(* PLC project machine, CODESYS STW CODESYS V3.5 SP11 - ESX-3CS, author isoloader *)
(* stored: creationDateTime 2026-05-19T11:34:01.4368509, version 0.1, modificationDateTime 2026-01-26T17:08:03, organization Isoloader *)
(* isoloader machine - common to both plc and secondary devices *)

(* {attribute 'qualified_only'} *)
TYPE t_pack_code : (cPackCodeNone := 0, cPackCodeSystem := 1, cPackCodeMovement := 2, cPackCodeReportable := 3, cPackCodeSpreader := 4, cPackCodeConfiguration := 5, cPackCodeUICommand := 6);
END_TYPE

FUNCTION_BLOCK PackChannelUInterface EXTENDS NonOperationalParticleSet
  VAR
    lPLCIncomingChannel : PackChannel;
    lPLCOutgoingChannel : PackChannel;
    lPLCOutgoingPacket : t_packet;
    lPLCIncomingPacket : t_packet;
    lDebugPack : BOOL := FALSE;
    lDebugUnpack : BOOL := FALSE;
    lDebugPackPacket : t_packet;
    lDebugUnpackPacket : t_packet;
    lPackTimer : t_timer;
    lPackSystem : REFERENCE TO PackSystem;
    lPackMovement : REFERENCE TO PackMovement;
    lPackReportable : REFERENCE TO PackReportable;
    lPackSpreader : REFERENCE TO PackSpreader;
    lPackUICommand : REFERENCE TO PackUICommand;
    lPackProvider : REFERENCE TO PackProvider;
  END_VAR

            ;
          

METHOD initialize
                  IF ((NOT(__ISVALIDREF(lPackSystem))) OR
	(NOT(__ISVALIDREF(lPackMovement))) OR
	(NOT(__ISVALIDREF(lPackReportable))) OR
	(NOT(__ISVALIDREF(lPackSpreader))) OR
	(NOT(__ISVALIDREF(lPackUICommand))) OR
	(NOT(__ISVALIDREF(lPackProvider)))) THEN
	gCodeErrorHandler(pMessage:=CONCAT('null reference in ',lIdentity));
END_IF
	
lPackTimer.lEnable := TRUE;
lPackTimer.lPeriod := T#60MS;
lPackTimer.initialize();

lPLCOutgoingChannel.register(ADR(lPackSystem)); // foobar particle reorganization
lPLCOutgoingChannel.register(ADR(lPackMovement));
lPLCOutgoingChannel.register(ADR(lPackReportable));
lPLCOutgoingChannel.register(ADR(lPackSpreader));
lPLCOutgoingChannel.initialize();

lPLCIncomingChannel.register(ADR(lPackUICommand));
lPLCIncomingChannel.initialize();

SUPER^.initialize();
                
END_METHOD

METHOD initializePackChannelUInterface
  VAR_INPUT
    packSystem : REFERENCE TO PackSystem;
    packMovement : REFERENCE TO PackMovement;
    packReportable : REFERENCE TO PackReportable;
    packSpreader : REFERENCE TO PackSpreader;
    packUICommand : REFERENCE TO PackUICommand;
    packProvider : REFERENCE TO PackProvider;
  END_VAR
                  lPackSystem REF= packSystem;
lPackMovement REF= packMovement;
lPackReportable REF= packReportable;
lPackSpreader REF= packSpreader;

lPackUICommand REF= packUICommand;

lPackProvider REF= packProvider;

                
END_METHOD

METHOD trigger : BOOL
  VAR_INPUT
    machineStateId : t_machine_state_id;
  END_VAR
                  lPLCOutgoingChannel.trigger(lPLCOutgoingPacket,machineStateId);

                
END_METHOD

PROPERTY PackMovement : REFERENCE TO PackMovement
GET
                    PackMovement ref= lPackMovement;
                  
END_GET
END_PROPERTY

PROPERTY PackReportable : REFERENCE TO PackReportable
GET
                    PackReportable ref= lPackReportable;
                  
END_GET
END_PROPERTY

PROPERTY PackSpreader : REFERENCE TO PackSpreader
GET
                    PackSpreader ref= lPackSpreader;
                  
END_GET
END_PROPERTY

PROPERTY PackSystem : REFERENCE TO PackSystem
GET
                    PackSystem ref= lPackSystem;
                  
END_GET
END_PROPERTY

PROPERTY PackUICommand : REFERENCE TO PackUICommand
GET
                    PackUICommand ref= lPackUICommand;
                  
END_GET
END_PROPERTY

PROPERTY TypeToken : t_medium_string
GET
                    TypeToken := 'PackChannelUI';
                  
END_GET
END_PROPERTY
END_FUNCTION_BLOCK

FUNCTION_BLOCK PackChannelUInterfacePLC EXTENDS PackChannelUInterface

            ;
          

METHOD pullPLCIncomingChannel : BOOL
                  pullPLCIncomingChannel := FALSE;

lPackProvider.pull();

IF (lPLCIncomingPacket.Byte1<>lPackProvider.PackIn1) THEN
	lPLCIncomingPacket.Byte1 := lPackProvider.PackIn1;
	lPLCIncomingPacket.Byte1 := lPLCIncomingPacket.Byte1 OR INT_TO_USINT(cPackCodeUICommand);
	gSystemPrimary.Active.registerUI();
	pullPLCIncomingChannel := TRUE;
END_IF

IF (lPLCIncomingPacket.Byte2<>lPackProvider.PackIn2) THEN
	lPLCIncomingPacket.Byte2 := lPackProvider.PackIn2;
	gSystemPrimary.Active.registerUI();
	pullPLCIncomingChannel := TRUE;
END_IF

IF (lPLCIncomingPacket.Byte3<>lPackProvider.PackIn3) THEN
	lPLCIncomingPacket.Byte3 := lPackProvider.PackIn3;
	gSystemPrimary.Active.registerUI();
	pullPLCIncomingChannel := TRUE;
END_IF

IF (lPLCIncomingPacket.Byte4<>lPackProvider.PackIn4) THEN
	lPLCIncomingPacket.Byte4 := lPackProvider.PackIn4;
	gSystemPrimary.Active.registerUI();
	pullPLCIncomingChannel := TRUE;
END_IF

IF (lPLCIncomingPacket.Byte5<>lPackProvider.PackIn5) THEN
	lPLCIncomingPacket.Byte5 := lPackProvider.PackIn5;
	gSystemPrimary.Active.registerUI();
	pullPLCIncomingChannel := TRUE;
END_IF

IF (lPLCIncomingPacket.Byte6<>lPackProvider.PackIn6) THEN
	lPLCIncomingPacket.Byte6 := lPackProvider.PackIn6;
	gSystemPrimary.Active.registerUI();
	pullPLCIncomingChannel := TRUE;
END_IF

IF (lPLCIncomingPacket.Byte7<>lPackProvider.PackIn7) THEN
	lPLCIncomingPacket.Byte7 := lPackProvider.PackIn7;
	gSystemPrimary.Active.registerUI();
	pullPLCIncomingChannel := TRUE;
END_IF

IF (lPLCIncomingPacket.Byte8<>lPackProvider.PackIn8) THEN
	lPLCIncomingPacket.Byte8 := lPackProvider.PackIn8;
	gSystemPrimary.Active.registerUI();
	pullPLCIncomingChannel := TRUE;
END_IF

                
END_METHOD

METHOD pushPLCOutgoingChannel
                  lPackProvider.PackOut1 := lPLCOutgoingPacket.Byte1;
lPackProvider.PackOut2 := lPLCOutgoingPacket.Byte2;
lPackProvider.PackOut3 := lPLCOutgoingPacket.Byte3;
lPackProvider.PackOut4 := lPLCOutgoingPacket.Byte4;
lPackProvider.PackOut5 := lPLCOutgoingPacket.Byte5;
lPackProvider.PackOut6 := lPLCOutgoingPacket.Byte6;
lPackProvider.PackOut7 := lPLCOutgoingPacket.Byte7;
lPackProvider.PackOut8 := lPLCOutgoingPacket.Byte8;

lPackProvider.push();

                
END_METHOD

METHOD operator
                  lPackTimer.operator();
IF ((NOT(lPackTimer.Enable)) OR (lPackTimer.Expired)) THEN
	lPackTimer.reset();

	lPLCOutgoingChannel.pack(lPLCOutgoingPacket);
	pushPLCOutgoingChannel();
			
	IF (lDebugPack) THEN
		lDebugPackPacket.copy(lPLCOutgoingPacket);
	END_IF
END_IF

IF (pullPLCIncomingChannel()) THEN
	IF (lDebugUnpack) THEN
		lDebugUnpackPacket.copy(lPLCIncomingPacket);
	END_IF

	lPLCIncomingChannel.unpack(lPLCIncomingPacket);
END_IF

                
END_METHOD
END_FUNCTION_BLOCK

FUNCTION_BLOCK PackMovement EXTENDS Packer
  VAR_INPUT
    lSteerStateA : t_adjust_state;
    lSteerStateB : t_adjust_state;
    lSteerStateC : t_adjust_state;
    lSteerStateD : t_adjust_state;
    lSteerTargetAngle : REAL;
    lSteerCurrentMode : t_steer_mode;
    lTravelActive : BOOL;
    lTravelVelocity : t_percentage;
    lLiftActive : BOOL;
    lLiftABPosition : t_percentage;
    lLiftCDPosition : t_percentage;
    lProgrammedMovementCurrent : t_prog_mov_code;
    lProgrammedMovementState : t_prog_mov_state;
  END_VAR

            
          

METHOD _unpack
  VAR_INPUT
    packet : REFERENCE TO t_packet;
  END_VAR
                  lSteerStateA := packet.unpackUSINT(5,3);
lSteerStateB := packet.unpackUSINT(8,3);
lSteerStateC := packet.unpackUSINT(11,3);
lSteerStateD := packet.unpackUSINT(14,3);

lSteerTargetAngle := AngleFromSINT(packet.unpackSINT(17,8));
lSteerCurrentMode := USINT_TO_INT(packet.unpackUSINT(25,4));

lTravelActive := packet.unpackBool(29);
lTravelVelocity :=  SignedPercentageFrom6bits(packet.unpackUSINT(30,6));

lLiftActive := packet.unpackBool(36);
lLiftABPosition := SignedPercentageFrom7bits(packet.unpackUSINT(37,7));
lLiftCDPosition := SignedPercentageFrom7bits(packet.unpackUSINT(44,7));

lProgrammedMovementCurrent := packet.unpackUSINT(51,5);
lProgrammedMovementState := packet.unpackUSINT(56,3);
                
END_METHOD

METHOD _pack
  VAR_INPUT
    packet : REFERENCE TO t_packet;
  END_VAR
                  packet.packUSINT(INT_TO_USINT(lSteerStateA),5,3);
packet.packUSINT(INT_TO_USINT(lSteerStateB),8,3);
packet.packUSINT(INT_TO_USINT(lSteerStateC),11,3);
packet.packUSINT(INT_TO_USINT(lSteerStateD),14,3);

packet.packSINT(AngleAsSINT(lSteerTargetAngle),17,8);
packet.packUSINT(INT_TO_USINT(lSteerCurrentMode),25,4);

packet.packBool(lTravelActive,29);
packet.packUSINT(SignedPercentageAs6bits(lTravelVelocity),30,6);

packet.packBool(lLiftActive,36);
packet.packUSINT(SignedPercentageAs7bits(lLiftABPosition),37,7);
packet.packUSINT(SignedPercentageAs7bits(lLiftCDPosition),44,7);

packet.packUSINT(INT_TO_USINT(lProgrammedMovementCurrent),51,5);
packet.packUSINT(INT_TO_USINT(lProgrammedMovementState),56,3);

                
END_METHOD

METHOD initialize
                  lCode := INT_TO_USINT(t_pack_code.cPackCodeMovement);

SUPER^.initialize();

                
END_METHOD
END_FUNCTION_BLOCK

FUNCTION_BLOCK PackReportable EXTENDS Packer
  VAR_INPUT
    lReportableA : t_ui_reportable;
    lReportableB : t_ui_reportable;
    lReportableC : t_ui_reportable;
    lReportableD : t_ui_reportable;
  END_VAR

            
          

METHOD _unpack
  VAR_INPUT
    packet : REFERENCE TO t_packet;
  END_VAR
  VAR
    b : BOOL;
  END_VAR
                  IF (packet.unpackBool(5)) THEN
	lReportableA.valid := TRUE;
	lReportableA.state := packet.unpackUSINT(6,8);
ELSE
	lReportableA.event := packet.unpackUSINT(6,8);
	IF (lReportableA.event=cECNone) THEN
		lReportableA.valid := FALSE;
		lReportableB.valid := FALSE;
		lReportableC.valid := FALSE;
		lReportableD.valid := FALSE;
		
		RETURN;				
	END_IF
	lReportableA.valid := TRUE;
END_IF
lReportableA.active := packet.unpackBool(14);
lReportableA.subsystem := packet.unpackUSINT(15,5);

IF (packet.unpackBool(20)) THEN
	lReportableB.valid := TRUE;
	lReportableB.state := packet.unpackUSINT(21,8);
ELSE
	lReportableB.event := packet.unpackUSINT(21,8);	
	IF (lReportableB.event=cECNone) THEN
		lReportableB.valid := FALSE;
		lReportableC.valid := FALSE;
		lReportableD.valid := FALSE;
		
		RETURN;				
	END_IF
	lReportableB.valid := TRUE;
END_IF
lReportableB.active := packet.unpackBool(29);
lReportableB.subsystem := packet.unpackUSINT(30,5);

IF (packet.unpackBool(35)) THEN
	lReportableC.valid := TRUE;
	lReportableC.state := packet.unpackUSINT(36,8);
ELSE
	lReportableC.event := packet.unpackUSINT(36,8);	
	IF (lReportableC.event=cECNone) THEN
		lReportableC.valid := FALSE;
		lReportableD.valid := FALSE;
		
		RETURN;				
	END_IF
	lReportableC.valid := TRUE;
END_IF
lReportableC.active := packet.unpackBool(44);
lReportableC.subsystem := packet.unpackUSINT(45,5);

IF (packet.unpackBool(50)) THEN
	lReportableD.valid := TRUE;
	lReportableD.state := packet.unpackUSINT(51,8);
ELSE
	lReportableD.event := packet.unpackUSINT(51,8);	
	IF (lReportableD.event=cECNone) THEN
		lReportableD.valid := FALSE;
		
		RETURN;				
	END_IF
	lReportableD.valid := TRUE;
END_IF
lReportableD.active := packet.unpackBool(59);
lReportableD.subsystem := packet.unpackUSINT(60,5);

                
END_METHOD

METHOD _pack
  VAR_INPUT
    packet : REFERENCE TO t_packet;
  END_VAR
                  IF (NOT(lReportableA.valid)) THEN
	RETURN;
END_IF
	
IF (lReportableA.event=cECNone) THEN
	packet.packBool(TRUE,5);
	packet.packUSINT(INT_TO_USINT(lReportableA.state),6,8);
ELSE
	packet.packBool(FALSE,5);
	packet.packUSINT(INT_TO_USINT(lReportableA.event),6,8);
END_IF
packet.packBool(lReportableA.active,14);
packet.packUSINT(INT_TO_USINT(lReportableA.subsystem),15,5);

IF (NOT(lReportableB.valid)) THEN
	RETURN;
END_IF

IF (lReportableB.event=cECNone) THEN
	packet.packBool(TRUE,20);
	packet.packUSINT(INT_TO_USINT(lReportableB.state),21,8);
ELSE
	packet.packBool(FALSE,20);
	packet.packUSINT(INT_TO_USINT(lReportableB.event),21,8);
END_IF
packet.packBool(lReportableB.active,29);
packet.packUSINT(INT_TO_USINT(lReportableB.subsystem),30,5);

IF (NOT(lReportableC.valid)) THEN
	RETURN;
END_IF

IF (lReportableC.event=cECNone) THEN
	packet.packBool(TRUE,35);
	packet.packUSINT(INT_TO_USINT(lReportableC.state),36,8);
ELSE
	packet.packBool(FALSE,35);
	packet.packUSINT(INT_TO_USINT(lReportableC.event),36,8);
END_IF
packet.packBool(lReportableC.active,44);
packet.packUSINT(INT_TO_USINT(lReportableC.subsystem),45,5);

IF (NOT(lReportableD.valid)) THEN
	RETURN;
END_IF

IF (lReportableD.event=cECNone) THEN
	packet.packBool(TRUE,50);
	packet.packUSINT(INT_TO_USINT(lReportableD.state),51,8);
ELSE
	packet.packBool(FALSE,50);
	packet.packUSINT(INT_TO_USINT(lReportableD.event),51,8);
END_IF
packet.packBool(lReportableD.active,59);
packet.packUSINT(INT_TO_USINT(lReportableD.subsystem),60,5);

                
END_METHOD

METHOD initialize
                  lCode := INT_TO_USINT(t_pack_code.cPackCodeReportable);

SUPER^.initialize();

                
END_METHOD

METHOD reset
                  SUPER^.reset();

lReportableA.valid := FALSE;
lReportableB.valid := FALSE;
lReportableC.valid := FALSE;
lReportableD.valid := FALSE;
                
END_METHOD
END_FUNCTION_BLOCK

FUNCTION_BLOCK PackSpreader EXTENDS Packer
  VAR_INPUT
    lSideShiftActive : BOOL;
    lTwistlocksState : t_lock_state;
    lStateA : t_lock_state;
    lLoweredA : BOOL;
    lStateB : t_lock_state;
    lLoweredB : BOOL;
    lStateC : t_lock_state;
    lLoweredC : BOOL;
    lStateD : t_lock_state;
    lLoweredD : BOOL;
    lExtensionState : t_spreader_extension_state;
    lSpreaderOperationEnabled : BOOL;
    lSpreaderOperationActive : BOOL;
    lSpreaderConfigurationOptionEnabled : BOOL;
    lSpreaderConfigurationEnabled : BOOL;
    lSpreaderConfigurationActive : BOOL;
    lSpreaderConfigurationExtending : BOOL;
    lSpreaderConfigurationRetracting : BOOL;
    lTopbeamActive : BOOL;
    lTopbeamABPosition : t_percentage;
    lTopbeamCDPosition : t_percentage;
  END_VAR

            
          

METHOD _unpack
  VAR_INPUT
    packet : REFERENCE TO t_packet;
  END_VAR
                  lSideShiftActive := packet.unpackBool(5);

lTwistlocksState := packet.unpackUSINT(6,2);

lStateA := packet.unpackUSINT(8,2);
lLoweredA := packet.unpackBool(10);
lStateB := packet.unpackUSINT(11,2);
lLoweredB := packet.unpackBool(13);
lStateC := packet.unpackUSINT(14,2);
lLoweredC := packet.unpackBool(16);
lStateD := packet.unpackUSINT(17,2);
lLoweredD := packet.unpackBool(19);

lExtensionState := packet.unpackUSINT(20,2);
lSpreaderOperationEnabled := packet.unpackBool(22);
lSpreaderOperationActive := packet.unpackBool(23);

lSpreaderConfigurationOptionEnabled := packet.unpackBool(24);
lSpreaderConfigurationEnabled := packet.unpackBool(25);
lSpreaderConfigurationActive := packet.unpackBool(26);
lSpreaderConfigurationExtending := packet.unpackBool(27);
lSpreaderConfigurationRetracting := packet.unpackBool(28);

lTopbeamActive := packet.unpackBool(29);
lTopbeamABPosition := SignedPercentageFrom7bits(packet.unpackUSINT(30,7));
lTopbeamCDPosition := SignedPercentageFrom7bits(packet.unpackUSINT(37,7));


                
END_METHOD

METHOD _pack
  VAR_INPUT
    packet : REFERENCE TO t_packet;
  END_VAR
                  packet.packBool(lSideShiftActive,5);

//6-32 27 bits

packet.packUSINT(INT_TO_USINT(lTwistlocksState),6,2);

packet.packUSINT(INT_TO_USINT(lStateA),8,2);
packet.packBool(lLoweredA,10);
packet.packUSINT(INT_TO_USINT(lStateB),11,2);
packet.packBool(lLoweredB,13);
packet.packUSINT(INT_TO_USINT(lStateC),14,2);
packet.packBool(lLoweredC,16);
packet.packUSINT(INT_TO_USINT(lStateD),17,2);
packet.packBool(lLoweredD,19);

packet.packUSINT(INT_TO_USINT(lExtensionState),20,2);
packet.packBool(lSpreaderOperationEnabled,22);
packet.packBool(lSpreaderOperationActive,23);

packet.packBool(lSpreaderConfigurationOptionEnabled,24);
packet.packBool(lSpreaderConfigurationEnabled,25);
packet.packBool(lSpreaderConfigurationActive,26);
packet.packBool(lSpreaderConfigurationExtending,27);
packet.packBool(lSpreaderConfigurationRetracting,28);

packet.packBool(lTopbeamActive,29);
packet.packUSINT(SignedPercentageAs7bits(lTopbeamABPosition),30,7);
packet.packUSINT(SignedPercentageAs7bits(lTopbeamCDPosition),37,7);


                
END_METHOD

METHOD initialize
                  lCode := INT_TO_USINT(t_pack_code.cPackCodeSpreader);

SUPER^.initialize();
                
END_METHOD
END_FUNCTION_BLOCK

FUNCTION_BLOCK PackSystem EXTENDS Packer
  VAR_INPUT
    lFunctionalMode : t_functional_mode;
    lToggle : BOOL;
    lSystemState : t_system_state;
    lOperatingMode : t_operating_mode;
    lSpeedModeSlow : BOOL;
    lLightStatus : BOOL;
    lUIReady : BOOL;
    lUIModeRequest : BOOL;
    lUIMode : t_ui_mode;
    lHours : UINT;
    lSOC : t_percentage;
    lCurrent : t_percentage;
    lInputMode : t_input_mode;
    lUIOrientation : t_ui_orientation;
    lAvailability : t_percentage;
  END_VAR
  VAR
    lOverrideSystemState : BOOL := FALSE;
    lOverrideSystemStateValue : t_system_state := cSystemStateOperational;
  END_VAR

            
          

METHOD _unpack
  VAR_INPUT
    packet : REFERENCE TO t_packet;
  END_VAR
                  lFunctionalMode := packet.unpackUSINT(5,3);
lToggle := packet.unpackBool(8);
lSystemState := packet.unpackUSINT(9,4);
lOperatingMode := packet.unpackUSINT(13,4);
lSpeedModeSlow := packet.unpackBool(17);
lLightStatus := packet.unpackBool(18);
lUIReady := packet.unpackBool(19);
lUIModeRequest := packet.unpackBool(20);
lUIMode := packet.unpackUSINT(21,2);
lHours := packet.unpackUINT(23,16);
lSOC := PercentageFrom7bits(packet.unpackUSINT(39,7));
lCurrent := SignedPercentageFrom8bits(packet.unpackUSINT(46,8));
lInputMode := packet.unpackUSINT(54,2);
lUIOrientation := packet.unpackUSINT(56,3);
lAvailability := PercentageFrom4bits(packet.unpackUSINT(59,4));

IF (lOverrideSystemState) THEN
	lSystemState := lOverrideSystemStateValue;
END_IF


                
END_METHOD

METHOD _pack
  VAR_INPUT
    packet : REFERENCE TO t_packet;
  END_VAR
                  packet.packUSINT(INT_TO_USINT(lFunctionalMode),5,3);
packet.packBool(lToggle,8);
packet.packUSINT(INT_TO_USINT(lSystemState),9,4);
packet.packUSINT(INT_TO_USINT(lOperatingMode),13,4);
packet.packBool(lSpeedModeSlow,17);
packet.packBool(lLightStatus,18);
packet.packBool(lUIReady,19);
packet.packBool(lUIModeRequest,20);
packet.packUSINT(INT_TO_USINT(lUIMode),21,2);
packet.packUINT(lHours,23,16);
packet.packUSINT(PercentageAs7bits(lSOC),39,7);
packet.packUSINT(SignedPercentageAs8bits(lCurrent),46,8);
packet.packUSINT(INT_TO_USINT(lInputMode),54,2);
packet.packUSINT(INT_TO_USINT(lUIOrientation),56,3);
packet.packUSINT(PercentageAs4bits(lAvailability),59,4);

                
END_METHOD

METHOD initialize
                  lCode := INT_TO_USINT(t_pack_code.cPackCodeSystem);

SUPER^.initialize();



                
END_METHOD
END_FUNCTION_BLOCK

FUNCTION_BLOCK PackUICommand EXTENDS Packer
  VAR_INPUT
    lUIModeResponse : BOOL;
    lUIEventCodeRequest : t_ui_event_code;
    lSteerModeRequest : t_steer_mode;
    lOperatingMethodRequest : t_operating_method;
    lFunctionalModeRequest : t_functional_mode;
    lInputModeRequest : t_input_mode;
    lUIOrientationRequest : t_ui_orientation;
    lAutomationRequest : t_prog_mov_code;
    lIsBeginner : BOOL;
    lOverride : BOOL;
    lReportableA : t_ui_reportable;
    lReportableB : t_ui_reportable;
  END_VAR
  VAR
    lTimer : t_timer;
  END_VAR

            
          

METHOD reset
                  SUPER^.reset();

lUIModeResponse := FALSE;
lUIEventCodeRequest := cUIEventCodeNone;
lSteerModeRequest := cSteerModeNone;
lOperatingMethodRequest := cOperatingMethodNone;
lFunctionalModeRequest := cFunctionalModeAny;
lInputModeRequest := cInputModeNone;
lAutomationRequest := cProgMovCodeNone;
lIsBeginner := FALSE;

lReportableA.valid := FALSE;
lReportableB.valid := FALSE;


                
END_METHOD

METHOD trigger : BOOL
  VAR_INPUT
    packet : REFERENCE TO t_packet;
    machineStateId : t_machine_state_id;
  END_VAR
                  trigger := TRUE;
(*
CASE machineStateId OF
	t_machine_state_id.cMSIdNone:
		RETURN;

	t_machine_state_id.cMSIdSteerModeRequest:
		lTimer.reset();		
		packet.packUSINT(INT_TO_USINT(lPackRadioDashboard.lSteerModeRequest),14,3);
		RETURN;

	t_machine_state_id.cMSIdSteerModeRequest4WS:
		lTimer.reset();		
		packet.packUSINT(INT_TO_USINT(t_steer_mode.cSteerMode4WS),14,3);
		RETURN;

	t_machine_state_id.cMSIdSteerModeRequestLateral:
		lTimer.reset();		
		packet.packUSINT(INT_TO_USINT(t_steer_mode.cSteerModeLateral),14,3);
		RETURN;

	t_machine_state_id.cMSIdSteerModeRequestCarousel:
		lTimer.reset();		
		packet.packUSINT(INT_TO_USINT(t_steer_mode.cSteerModeCarousel),14,3);
		RETURN;

	
	t_machine_state_id.cMSIdToggleLightsRequest:
		lTimer.reset();
		packet.packUSINT(INT_TO_USINT(t_ui_event_code.cUIEventCodeToggleLights),8,6);
		RETURN;
	
	t_machine_state_id.cMSIdRadioModeResponse:
		lTimer.reset();
		packet.packUSINT(INT_TO_USINT(t_ui_event_code.cUIEventCodeUIModeResponse),8,6);		
		RETURN;
		
	t_machine_state_id.cMSIdOperatingModeRequest:
		lTimer.reset();		
		packet.packUSINT(INT_TO_USINT(lPackRadioDashboard.lOperatingMethodRequest),17,3);	
		RETURN;

	t_machine_state_id.cMSIdSpreaderTelescopingExtensionStateRequest6m:
		lTimer.reset();		
		packet.packUSINT(INT_TO_USINT(t_spreader_extension_state.cSpreaderExtensionState6m),20,2);
		RETURN;
	
	t_machine_state_id.cMSIdSpreaderTelescopingExtensionStateRequest9m:
		lTimer.reset();		
		packet.packUSINT(INT_TO_USINT(t_spreader_extension_state.cSpreaderExtensionState9m),20,2);
		RETURN;
		
	t_machine_state_id.cMSIdSpreaderTelescopingExtensionStateRequest12m:
		lTimer.reset();		
		packet.packUSINT(INT_TO_USINT(t_spreader_extension_state.cSpreaderExtensionState12m),20,2);
		RETURN;

	t_machine_state_id.cMSIdSpreaderGrabArmsExtendABRequest:
		lTimer.reset();		
		packet.packUSINT(INT_TO_USINT(t_spreader_extension_method.cSpreaderExtensionMethodABExtend),22,3);
		RETURN;

	t_machine_state_id.cMSIdSpreaderGrabArmsRetractABRequest:
		lTimer.reset();		
		packet.packUSINT(INT_TO_USINT(t_spreader_extension_method.cSpreaderExtensionMethodABRetract),22,3);	
		RETURN;

	t_machine_state_id.cMSIdSpreaderGrabArmsExtendCDRequest:
		lTimer.reset();		
		packet.packUSINT(INT_TO_USINT(t_spreader_extension_method.cSpreaderExtensionMethodCDExtend),22,3);	
		RETURN;

	t_machine_state_id.cMSIdSpreaderGrabArmsRetractCDRequest:
		lTimer.reset();		
		packet.packUSINT(INT_TO_USINT(t_spreader_extension_method.cSpreaderExtensionMethodCDRetract),22,3);		
		RETURN;
		
	t_machine_state_id.cMSIdLiftTopRequest:
		lTimer.reset();
		packet.packUSINT(INT_TO_USINT(t_ui_event_code.cUIEventCodeLiftTop),8,6);
		RETURN;	
		
END_CASE
*)
trigger := FALSE;

                
END_METHOD

METHOD _unpack
  VAR_INPUT
    packet : REFERENCE TO t_packet;
  END_VAR
                  lUIModeResponse := packet.unpackBool(5);
lUIEventCodeRequest := packet.unpackUSINT(6,6);
lSteerModeRequest := packet.unpackUSINT(12,3);
lOperatingMethodRequest := packet.unpackUSINT(15,3);
lFunctionalModeRequest := packet.unpackUSINT(18,3);
lInputModeRequest := packet.unpackUSINT(21,2);
lUIOrientationRequest := packet.unpackUSINT(23,3);
lAutomationRequest := packet.unpackUSINT(26,5);
lIsBeginner := packet.unpackBool(31);
lOverride := packet.unpackBool(32);

IF (packet.unpackBool(33)) THEN
	lReportableA.valid := TRUE;
	lReportableA.state := packet.unpackUSINT(34,8);
ELSE
	lReportableA.event := packet.unpackUSINT(34,8);
	IF (lReportableA.event=cECNone) THEN
		lReportableA.valid := FALSE;
		lReportableB.valid := FALSE;
		
		RETURN;				
	END_IF
	lReportableA.valid := TRUE;
END_IF
lReportableA.active := packet.unpackBool(42);
lReportableA.subsystem := packet.unpackUSINT(43,5);

IF (packet.unpackBool(49)) THEN
	lReportableB.valid := TRUE;
	lReportableB.state := packet.unpackUSINT(50,8);
ELSE
	lReportableB.event := packet.unpackUSINT(50,8);	
	IF (lReportableB.event=cECNone) THEN
		lReportableB.valid := FALSE;
		
		RETURN;				
	END_IF
	lReportableB.valid := TRUE;
END_IF
lReportableB.active := packet.unpackBool(58);
lReportableB.subsystem := packet.unpackUSINT(59,5);

                
END_METHOD

METHOD initialize
                  lCode := INT_TO_USINT(t_pack_code.cPackCodeUICommand);

SUPER^.initialize();

lTimer.initialize();
lTimer.Enable := TRUE;
lTimer.Period := T#60MS;


                
END_METHOD

METHOD _pack
  VAR_INPUT
    packet : REFERENCE TO t_packet;
  END_VAR
                  packet.packBool(lUIModeResponse,5);
packet.packUSINT(INT_TO_USINT(lUIEventCodeRequest),6,6);
packet.packUSINT(INT_TO_USINT(lSteerModeRequest),12,3);
packet.packUSINT(INT_TO_USINT(lOperatingMethodRequest),15,3);
packet.packUSINT(INT_TO_USINT(lFunctionalModeRequest),18,3);
packet.packUSINT(INT_TO_USINT(lInputModeRequest),21,2);
packet.packUSINT(INT_TO_USINT(lUIOrientationRequest),23,3);
packet.packUSINT(INT_TO_USINT(lAutomationRequest),26,5);
packet.packBool(lIsBeginner,31);
packet.packBool(lOverride,32);

IF (NOT(lReportableA.valid)) THEN
	RETURN;
END_IF
	
IF (lReportableA.event=cECNone) THEN
	packet.packBool(TRUE,33);
	packet.packUSINT(INT_TO_USINT(lReportableA.state),34,8);
ELSE
	packet.packBool(FALSE,33);
	packet.packUSINT(INT_TO_USINT(lReportableA.event),34,8);
END_IF
packet.packBool(lReportableA.active,42);
packet.packUSINT(INT_TO_USINT(lReportableA.subsystem),43,5);

IF (NOT(lReportableB.valid)) THEN
	RETURN;
END_IF
	
IF (lReportableB.event=cECNone) THEN
	packet.packBool(TRUE,49);
	packet.packUSINT(INT_TO_USINT(lReportableB.state),50,8);
ELSE
	packet.packBool(FALSE,49);
	packet.packUSINT(INT_TO_USINT(lReportableB.event),50,8);
END_IF
packet.packBool(lReportableB.active,58);
packet.packUSINT(INT_TO_USINT(lReportableB.subsystem),59,5);

                
END_METHOD
END_FUNCTION_BLOCK

FUNCTION_BLOCK PackProvider EXTENDS NonOperationalParticleSet
  VAR
    lPackIn1 : ValueObjectUSINTInputReferenceUSINT;
    lPackIn2 : ValueObjectUSINTInputReferenceUSINT;
    lPackIn3 : ValueObjectUSINTInputReferenceUSINT;
    lPackIn4 : ValueObjectUSINTInputReferenceUSINT;
    lPackIn5 : ValueObjectUSINTInputReferenceUSINT;
    lPackIn6 : ValueObjectUSINTInputReferenceUSINT;
    lPackIn7 : ValueObjectUSINTInputReferenceUSINT;
    lPackIn8 : ValueObjectUSINTInputReferenceUSINT;
    lPackOut1 : ValueObjectUSINTOutputReferenceUSINT;
    lPackOut2 : ValueObjectUSINTOutputReferenceUSINT;
    lPackOut3 : ValueObjectUSINTOutputReferenceUSINT;
    lPackOut4 : ValueObjectUSINTOutputReferenceUSINT;
    lPackOut5 : ValueObjectUSINTOutputReferenceUSINT;
    lPackOut6 : ValueObjectUSINTOutputReferenceUSINT;
    lPackOut7 : ValueObjectUSINTOutputReferenceUSINT;
    lPackOut8 : ValueObjectUSINTOutputReferenceUSINT;
  END_VAR

            ;
          

METHOD push
                  lPackOut1.operator();
lPackOut2.operator();
lPackOut3.operator();
lPackOut4.operator();
lPackOut5.operator();
lPackOut6.operator();
lPackOut7.operator();
lPackOut8.operator();

                
END_METHOD

METHOD pull
                  lPackIn1.operator();
lPackIn2.operator();
lPackIn3.operator();
lPackIn4.operator();
lPackIn5.operator();
lPackIn6.operator();
lPackIn7.operator();
lPackIn8.operator();

                
END_METHOD

METHOD initialize
                  lPackIn1.initializeValueObjectOp(NopSelf,'PackIn1','Packet 1 to master','',cValueStyleConfigurable);
lPackIn2.initializeValueObjectOp(NopSelf,'PackIn2','Packet 2 to master','',cValueStyleConfigurable);
lPackIn3.initializeValueObjectOp(NopSelf,'PackIn3','Packet 3 to master','',cValueStyleConfigurable);
lPackIn4.initializeValueObjectOp(NopSelf,'PackIn4','Packet 4 to master','',cValueStyleConfigurable);
lPackIn5.initializeValueObjectOp(NopSelf,'PackIn5','Packet 5 to master','',cValueStyleConfigurable);
lPackIn6.initializeValueObjectOp(NopSelf,'PackIn6','Packet 6 to master','',cValueStyleConfigurable);
lPackIn7.initializeValueObjectOp(NopSelf,'PackIn7','Packet 7 to master','',cValueStyleConfigurable);
lPackIn8.initializeValueObjectOp(NopSelf,'PackIn8','Packet 8 to master','',cValueStyleConfigurable);

lPackOut1.initializeValueObjectOp(NopSelf,'PackOut1','Packet 1 from master','',cValueStyleConfigurable);
lPackOut2.initializeValueObjectOp(NopSelf,'PackOut2','Packet 2 from master','',cValueStyleConfigurable);
lPackOut3.initializeValueObjectOp(NopSelf,'PackOut3','Packet 3 from master','',cValueStyleConfigurable);
lPackOut4.initializeValueObjectOp(NopSelf,'PackOut4','Packet 4 from master','',cValueStyleConfigurable);
lPackOut5.initializeValueObjectOp(NopSelf,'PackOut5','Packet 5 from master','',cValueStyleConfigurable);
lPackOut6.initializeValueObjectOp(NopSelf,'PackOut6','Packet 6 from master','',cValueStyleConfigurable);
lPackOut7.initializeValueObjectOp(NopSelf,'PackOut7','Packet 7 from master','',cValueStyleConfigurable);
lPackOut8.initializeValueObjectOp(NopSelf,'PackOut8','Packet 8 from master','',cValueStyleConfigurable);

SUPER^.initialize();
SubSystem := cSubsystemUInterface;

                
END_METHOD

METHOD initializePackProvider
  VAR_INPUT
    packIn1 : REFERENCE TO USINT;
    packIn2 : REFERENCE TO USINT;
    packIn3 : REFERENCE TO USINT;
    packIn4 : REFERENCE TO USINT;
    packIn5 : REFERENCE TO USINT;
    packIn6 : REFERENCE TO USINT;
    packIn7 : REFERENCE TO USINT;
    packIn8 : REFERENCE TO USINT;
    packOut1 : REFERENCE TO USINT;
    packOut2 : REFERENCE TO USINT;
    packOut3 : REFERENCE TO USINT;
    packOut4 : REFERENCE TO USINT;
    packOut5 : REFERENCE TO USINT;
    packOut6 : REFERENCE TO USINT;
    packOut7 : REFERENCE TO USINT;
    packOut8 : REFERENCE TO USINT;
  END_VAR
                  lPackIn1.InputReference REF= packIn1;
lPackIn2.InputReference REF= packIn2;
lPackIn3.InputReference REF= packIn3;
lPackIn4.InputReference REF= packIn4;
lPackIn5.InputReference REF= packIn5;
lPackIn6.InputReference REF= packIn6;
lPackIn7.InputReference REF= packIn7;
lPackIn8.InputReference REF= packIn8;

lPackOut1.OutputReference ref= packOut1;
lPackOut2.OutputReference ref= packOut2;
lPackOut3.OutputReference ref= packOut3;
lPackOut4.OutputReference ref= packOut4;
lPackOut5.OutputReference ref= packOut5;
lPackOut6.OutputReference ref= packOut6;
lPackOut7.OutputReference ref= packOut7;
lPackOut8.OutputReference ref= packOut8;

                
END_METHOD

PROPERTY PackIn1 : USINT
GET
                    PackIn1 := lPackIn1.Value;
                  
END_GET
END_PROPERTY

PROPERTY PackIn2 : USINT
GET
                    PackIn2 := lPackIn2.Value;
                  
END_GET
END_PROPERTY

PROPERTY PackIn3 : USINT
GET
                    PackIn3 := lPackIn3.Value;
                  
END_GET
END_PROPERTY

PROPERTY PackIn4 : USINT
GET
                    PackIn4 := lPackIn4.Value;
                  
END_GET
END_PROPERTY

PROPERTY PackIn5 : USINT
GET
                    PackIn5 := lPackIn5.Value;
                  
END_GET
END_PROPERTY

PROPERTY PackIn6 : USINT
GET
                    PackIn6 := lPackIn6.Value;
                  
END_GET
END_PROPERTY

PROPERTY PackOut1 : USINT
SET
                    lPackOut1.Value := PackOut1;
                  
END_SET
END_PROPERTY

PROPERTY PackOut2 : USINT
SET
                    lPackOut2.Value := PackOut2;
                  
END_SET
END_PROPERTY

PROPERTY PackOut3 : USINT
SET
                    lPackOut3.Value := PackOut3;
                  
END_SET
END_PROPERTY

PROPERTY PackOut4 : USINT
SET
                    lPackOut4.Value := PackOut4;
                  
END_SET
END_PROPERTY

PROPERTY PackOut5 : USINT
SET
                    lPackOut5.Value := PackOut5;
                  
END_SET
END_PROPERTY

PROPERTY PackOut6 : USINT
SET
                    lPackOut6.Value := PackOut6;
                  
END_SET
END_PROPERTY

PROPERTY PackOut7 : USINT
SET
                    lPackOut7.Value := PackOut7;
                  
END_SET
END_PROPERTY

PROPERTY PackOut8 : USINT
SET
                    lPackOut8.Value := PackOut8;
                  
END_SET
END_PROPERTY

PROPERTY PackIn7 : USINT
GET
                    PackIn7 := lPackIn7.Value;
                  
END_GET
END_PROPERTY

PROPERTY PackIn8 : USINT
GET
                    PackIn8 := lPackIn8.Value;
                  
END_GET
END_PROPERTY

PROPERTY TypeToken : t_medium_string
GET
                    TypeToken := 'PackProvider';
                  
END_GET
END_PROPERTY
END_FUNCTION_BLOCK
